// TIA Portal V19 export
DATA_BLOCK "PNDevDiagInterface"   // DB50
TITLE = DevDiagInterface
{ DB_Accessible_From_OPC_UA := 'FALSE' }
FAMILY : Diag
// Interface Profinet device diagnostic / Schnittstelle Profinet Device Diagnose
// stored: DBAccessibleFromOPCUA false, InstanceOfName LAF_typeDevDiagInterface, InstanceOfType UDT
"LAF_typeDevDiagInterface"
   // VAR
   //    globalInfoHmi : "LAF_typeDevDiagGlobal";
   //    devStateHmi { ExternalWritable := 'False'} : Array[0..256] of "LAF_typeDevDiagBasic";
   //    devStateUser { ExternalAccessible := 'False'; ExternalVisible := 'False'; ExternalWritable := 'False'} : Array[0..256] of "LAF_typeDevDiagState";
   // END_VAR
BEGIN
END_DATA_BLOCK
